{attribute 'GeneratedUsingTerminal: EK1100-0000-0018'}
{attribute addProperty BoxType "EK1100-0000-0018"}
{attribute addProperty Id "Beckhoff_EJ4xxxEK1122Beckhoff_EJ4xxxEK1122_0F216A002A_0001_EJ4002_0000_0017EJ4002_24FBDF2D15A_0002_EJ4002_0000_0018EJ4002_36452C7415A_0003_EJ4004_0000_0020EJ4004_F6F08E1219A_0004_EJ4008_0000_0020EJ4008_B54D005F27A_0005_EJ4018_0000_0016EJ4018_B54D005F27A_0006_EJ4024_0000_0020EJ4024_F6F08E1219A_0007_EJ4132_0000_0019EJ4132_24FBDF2D15A_0008_EJ4134_0000_0019EJ4134_C861457119A_0009_EJ4134_0000_0020EJ4134_C861457119"}
{attribute addProperty CRC "3720346385"}
{attribute addProperty Size "177"}
TYPE Beckhoff_EJ4xxx_DDBFFB11 EXTENDS EK1100_AB5A9467 :
STRUCT
	{attribute addProperty Name "Beckhoff_EJ4xxxEK1122"}
	Beckhoff_EJ4xxxEK1122 : Beckhoff_EJ4xxxEK1122_0F216A00;
	{attribute addProperty Name "A_0001_EJ4002_0000_0017"}
	A_0001_EJ4002_0000_0017 : EJ4002_24FBDF2D;
	{attribute addProperty Name "A_0002_EJ4002_0000_0018"}
	A_0002_EJ4002_0000_0018 : EJ4002_36452C74;
	{attribute addProperty Name "A_0003_EJ4004_0000_0020"}
	A_0003_EJ4004_0000_0020 : EJ4004_F6F08E12;
	{attribute addProperty Name "A_0004_EJ4008_0000_0020"}
	A_0004_EJ4008_0000_0020 : EJ4008_B54D005F;
	{attribute addProperty Name "A_0005_EJ4018_0000_0016"}
	A_0005_EJ4018_0000_0016 : EJ4018_B54D005F;
	{attribute addProperty Name "A_0006_EJ4024_0000_0020"}
	A_0006_EJ4024_0000_0020 : EJ4024_F6F08E12;
	{attribute addProperty Name "A_0007_EJ4132_0000_0019"}
	A_0007_EJ4132_0000_0019 : EJ4132_24FBDF2D;
	{attribute addProperty Name "A_0008_EJ4134_0000_0019"}
	A_0008_EJ4134_0000_0019 : EJ4134_C8614571;
	{attribute addProperty Name "A_0009_EJ4134_0000_0020"}
	A_0009_EJ4134_0000_0020 : EJ4134_C8614571;
END_STRUCT
END_TYPE

(* stored: Version 1.2.0.0, ProductVersion 3.1.4024.9
   DUT Beckhoff_EJ4xxx_DDBFFB11: Id {f857e8a8-d89d-47d0-91da-9e469427bd8a} *)
